{attribute 'linkalways'} 
{attribute 'no_explicit_call' := 'This FB is a CLASS and must be accessed using methods or properties'}
{attribute 'enable_dynamic_creation'}
FUNCTION_BLOCK _UINT EXTENDS NumericDatatypeBase
VAR
	localData : UINT;
	activeData : REFERENCE TO UINT REF= localData;
END_VAR

PROPERTY PUBLIC Address : PVOID
GET
Address := ADR(activeData);
END_GET
END_PROPERTY

METHOD PUBLIC ClearReference
VAR_INPUT
END_VAR
activeData REF= localData;
END_METHOD

METHOD PUBLIC Clone : I_Datatype
VAR
    pClone : POINTER TO _UINT;
END_VAR
pClone := __NEW(_UINT(InitialValue := Value));
Clone := pClone^;
END_METHOD

METHOD FB_init : BOOL
VAR_INPUT
	bInitRetains : BOOL; // if TRUE, the retain variables are initialized (warm start / cold start)
	bInCopyCode : BOOL;  // if TRUE, the instance afterwards gets moved into the copy code (online change)
	InitialValue : UINT;
END_VAR
localData := InitialValue;
END_METHOD

PROPERTY PUBLIC IsFloat : BOOL
GET
IsFloat := FALSE;
END_GET
END_PROPERTY

PROPERTY PUBLIC IsSigned : BOOL
GET
IsSigned := FALSE;
END_GET
END_PROPERTY

PROPERTY PUBLIC LowerBound : UINT
GET
LowerBound := DatatypeLimits.UINT_LOWER_LIMIT;
END_GET
END_PROPERTY

METHOD PUBLIC MakeReferenceTo
VAR_INPUT
	ReferenceTarget : REFERENCE TO UINT;
END_VAR
activeData REF= ReferenceTarget;
END_METHOD

PROPERTY PUBLIC Name : T_MAXSTRING
GET
Name := 'UINT';
END_GET
END_PROPERTY

METHOD PROTECTED SerializeLowerbound
VAR_INPUT
	Serializer : I_Serializer;
END_VAR
Serializer.AddUint(Lowerbound);
END_METHOD

METHOD PROTECTED SerializeUpperbound
VAR_INPUT
	Serializer : I_Serializer;
END_VAR
Serializer.AddUint(Upperbound);
END_METHOD

METHOD PUBLIC SerializeWith
VAR_INPUT
	Serializer : I_Serializer;
END_VAR
Serializer.AddUdint(activeData);
END_METHOD

PROPERTY PUBLIC Size : UDINT
GET
Size := SIZEOF(activeData);
END_GET
END_PROPERTY

METHOD TryDeserializeFrom : BOOL
VAR_INPUT
	Deserializer : I_Deserializer;
	Feedback : I_DeserializerFeedback;
END_VAR
TryDeserializeFrom := Deserializer.TryGetUint(activeData, Feedback);
END_METHOD

METHOD TryMakeReferenceTo : BOOL
VAR_INPUT
	Target : I_Datatype;
END_VAR
VAR
	pTargetData : POINTER TO UINT;
END_VAR
IF NOT (Target.Name = Name) THEN
	RETURN;
END_IF

pTargetData := Target.Address;
activeData REF= pTargetData^;
TryMakeReferenceTo := TRUE;
END_METHOD

PROPERTY PUBLIC UpperBound : UINT
GET
UpperBound :=  DatatypeLimits.UINT_UPPER_LIMIT;
END_GET
END_PROPERTY

PROPERTY PUBLIC Value : UINT
GET
Value := activeData;
END_GET
SET
activeData := Value;
END_SET
END_PROPERTY

END_FUNCTION_BLOCK

(* stored: Version 1.1.0.1, ProductVersion 3.1.4024.12
   POU _UINT: Id {995d668d-1756-0a37-2c05-8ca3ff4956f7}, SpecialFunc None
   Folder Constructor: Id {78aaa507-2df2-0e8f-2906-79584738539b}
   Folder Protected: Id {55a729f0-4ce5-0a78-0470-183bef3326ff}
   Property Address: Id {9113e6fc-4280-0ff4-3d2b-a83d2008abca}
   Get Get: Id {176769e7-8086-0d69-3e5d-cc926d7968c6}
   Method ClearReference: Id {9b81d0ba-9f4a-07df-2040-f46fe1d4bc71}
   Method Clone: Id {c8fd1376-1712-0dac-16c5-8905a47bb999}
   Method FB_init: Id {1b3dcef0-dbe1-0d86-2057-3a4715e36472}
   Property IsFloat: Id {7140672d-5959-0a51-3373-b65464df4977}
   Get Get: Id {fc679317-d1e9-0752-147c-8ed43b6b6b16}
   Property IsSigned: Id {3df495b6-39f4-0b06-15c5-d7569e99cc72}
   Get Get: Id {97002cca-10ef-09e2-3189-a072945bc5d6}
   Property LowerBound: Id {61a670fa-806e-03bc-2142-758f4fdad9d6}
   Get Get: Id {19efc0e2-5dce-0663-2c5c-58858e623cbd}
   Method MakeReferenceTo: Id {b10274ff-0b29-0b44-03ea-62adedeaede5}
   Property Name: Id {94757126-c5cf-0308-2a3a-6e739fa45cd7}
   Get Get: Id {3107bf3c-4784-022a-29d1-0abdeda9259a}
   Method SerializeLowerbound: Id {d8a973c7-48e2-00a7-3f38-25d8e310d7b2}
   Method SerializeUpperbound: Id {3122713b-7237-074c-2984-0b59a88cae91}
   Method SerializeWith: Id {494ad21a-65c8-05ba-2d20-49a40ad1e485}
   Property Size: Id {bfbaedb5-39cb-0dff-2817-b472e3637a30}
   Get Get: Id {471b7cef-513e-021b-21e7-0f34b9c19e18}
   Method TryDeserializeFrom: Id {e3b027be-e921-0b13-370d-c73573a548b2}
   Method TryMakeReferenceTo: Id {e28baef7-01df-036c-1fe8-8cd5a7847557}
   Property UpperBound: Id {070a80f1-5328-0bfc-2214-bd602f4bbaa7}
   Get Get: Id {5c065ea8-b4ad-0e82-184e-ec27fc9a72ef}
   Property Value: Id {b1f35337-325c-0c44-3636-76d1c7dc23dc}
   Get Get: Id {aef20d35-df0f-0e2d-2d4e-a345a0bb3ba7}
   Set Set: Id {713983f2-1711-0503-2fbb-063b619ce73b} *)
